TYPE ST_HmiCommunicationConfig :
STRUCT
    tWatchdogTimeout : TIME;
END_STRUCT
END_TYPE

(* stored: Version 1.1.0.1, ProductVersion 3.1.4026.20
   DUT ST_HmiCommunicationConfig: Id {72413807-3239-4fb4-8479-1f122fc4da96} *)
